// TIA Portal V20 export
TYPE "UDT_MotorData"
TITLE = UDT_MotorData
// stored: IsFailsafeCompliant false
   STRUCT
      Command : Bool;
      Feedback : Bool;
      Speed : Real;
      RunTime : DInt;
      FaultCode : Int;
   END_STRUCT;
END_TYPE
